TYPE
    TcoOscilatingConveyorFeeder_PlcToPc EXTENDS TcoCore.TcoStruct :
    STRUCT

        EntryFeederIsEmpty : BOOL;
        FlowSensor : BOOL;
        EntryFeederError : BOOL;
        ThrowBoxPresent : BOOL;
        OscConvError : BOOL;
        SideGuardAtHome : BOOL;
        SideGuardAtWork : BOOL;
        SafeCondition : BOOL;
        DoorOpen : BOOL;
        Mode : eCUMode;
        Config : TcoOscilatingConveyorFeeder_Config_v_1_x_x;
    END_STRUCT
END_TYPE

(* stored: Version 1.1.0.1
   DUT TcoOscilatingConveyorFeeder_PlcToPc: Id {8f188680-0707-4f07-a2fc-a268da38e12b} *)
